# EPICS StreamDevice protocol: apps/danfysikApp/Db/danfysik-8500.proto
OutTerminator = CR;
InTerminator = LF CR;

putInt    { out "\$1 %d"; }
putFloat  { out "\$1 %f"; }
putString { out "\$1 %s"; }
getInt    { out "\$1"; in "%d"; }
getFloat  { out "\$1"; in "%f"; }
getString { out "\$1"; in "%s"; }
